// TIA Portal V20 export
DATA_BLOCK "MotionNodes"   // DB313
// stored: Access Published, MemoryReserve 100, Namespace Unit1
   VAR
      MotionToPLC : "LER_typeMotionToPLC";
      PLCToMotion : "LER_typePLCToMotion";
   END_VAR
BEGIN
   // MotionToPLC.OutputInterface.FeedingRollerMove : Output Cam
   // MotionToPLC.OutputInterface.CutConveyorMove : Output Cam
   // MotionToPLC.OutputInterface.NGKickerMove : Output Cam
   // MotionToPLC.OutputInterface.PassKickerMove : Output Cam
   // MotionToPLC.OutputInterface.CutterMove : Output Cam
   // MotionToPLC.OutputInterface.AutoBusy : Motion Auto Busy
   // MotionToPLC.OutputInterface.AutoStandBy : Motion AutoStandBy(Wait)
   // PLCToMotion.Commands.Dancer.Enable : Command는 계속 살릴 필요 없음
   // PLCToMotion.Commands.ReelCutMain.OneCell : 원 피딩 명령 (탭정위치 잡기용)
   // PLCToMotion.Commands.ReelCutMain.FullStep : 전체 1Cycle
   // PLCToMotion.Commands.ReelCutMain.Auto : 전체 Auto
   // PLCToMotion.Commands.ReelCutMain.SemiStep : 컨베어 한피치 이동 명령 (리워크 + 잔량배출)
   // PLCToMotion.Commands.MeasureIMain.Enable : 상시로 True로 시켜놔야함
   // PLCToMotion.Parameter.ReelCutMain.OneCell.JogSpeed : 메뉴얼 동작이라서 조그 스피드로 돌음, 셀 정위치 잡는 용도라서 탭센서 감지 될때까지 구동함
   // PLCToMotion.Parameter.ReelCutMain.StepAuto.CellCount : 스택 둘중에 최소값 move
   // PLCToMotion.Parameter.ReelCutMain.StepAuto.MaxErrorCount : 미사용 할거임
   // PLCToMotion.Parameter.ReelCutMain.StepAuto.KickerDistance : 키커 한번 동작거리
   // PLCToMotion.Parameter.ReelCutMain.StepAuto.StackDelayLimit : Stack1StartRequest 또는 Stack2StartRequest 둘중 하나라도 True일때 딜레이 시간 이후에 출발할건지 값
   // PLCToMotion.Parameter.ReelCutMain.StepAuto.NoCutUse : 1= 컷팅 안한다, 0= 컷팅한다
   // PLCToMotion.Parameter.ReelCutMain.StepAuto.Stack1StartRequest : 스택 출발 요청 신호
   // PLCToMotion.Parameter.ReelCutMain.StepAuto.Stack2StartRequest : 스택 출발 요청 신호
   // PLCToMotion.Parameter.ReelCutMain.Calculate.CutterDistances : 커터 한번 동작 거리
   // PLCToMotion.Parameter.ReelCutMain.Calculate.VisionDistances : 비전 한번 동작거리
   // PLCToMotion.Parameter.ReelCutMain.Calculate.VisionTime : 비전 서보 다운후 대기 시간
   // PLCToMotion.Parameter.MeasureIMain.Tab.CutDistances : 탭센서 부터 커팅위치 까지 거리값
   // PLCToMotion.Parameter.MeasureIMain.Joint.JointFilterDistance : 이음매 테이프 센서 OnOff 최소 크기값(헌팅 방지용)
   // PLCToMotion.Parameter.MeasureIMain.Joint.JointSensorToCutDistance : 이음매 테이프 센서부터 커팅위치 거리값
   // PLCToMotion.Parameter.MeasureIMain.Cell.VisionUnUse : True = 비전 판정 데이터 안봄 (서보는 동작함)
   // PLCToMotion.Parameter.MeasureIMain.Cell.NGKickerUnUse : True = 무조건 PASS 키커로 침
   // PLCToMotion.Parameter.MeasureIMain.Cell.PassKickerUnUse : True = 무조건 NG 키커로 침
   // PLCToMotion.Parameter.MeasureIMain.Cell.AllNGMode : True = 샘플링 및 케파빌리티 용도
   // PLCToMotion.Parameter.MeasureIMain.Cell.CutToNgKickerDistance : 커팅위치 부터 NG 키커까지 거리 값
   // PLCToMotion.Parameter.MeasureIMain.Vision.VisionSensor : 실제 비전 센서
   // PLCToMotion.Parameter.MeasureIMain.Vision.VisionOK : 비전 판정
   // PLCToMotion.Parameter.MeasureIMain.Vision.VisionNG : 비전 판정
   // PLCToMotion.Parameter.MeasureIMain.Vision.CutToVisionSensorDistance : 커팅위치 부터 vision 센서까지 거리 값
   // PLCToMotion.Parameter.MeasureIMain.Vision.VisionTime : 비전 판정 대기시간 (시간 지나면 NG)
   // PLCToMotion.Parameter.MeasureIMain.NG.NGSensor : 실제 NG 키커 센서
   // PLCToMotion.Parameter.MeasureIMain.OK.OKSensor : 실제 Pass 키커 센서
END_DATA_BLOCK
